(*
SPDX-FileCopyrightText: © 2026 Oleksandr Tiutyk <trofimich@gmail.com>
SPDX-License-Identifier: MIT
License: https://opensource.org/license/mit
*)

(*!
<summary>
Beckhoff EL1004: 4-channel digital input terminal (24 V DC, 3 ms filter).
</summary>
<description>
Process image mapping structure for the EL1004 EtherCAT terminal with 4 discrete 24 V DC inputs.
When used for I/O, link located fields or their containing buffers to the matching selected PDOs.
The record is not a packed wire buffer; compiler padding is not part of the device specification.
Unlinked/default values do not prove valid I/O. The caller evaluates bus/channel validity before use.
Use one owner task per instance and externally synchronize other access; multi-field snapshots are not atomic.
Copies store data without creating hardware links. Keep borrowed field references valid while consumers are bound.
This passive record performs no validation, synchronization, configuration or protocol advancement.
</description>
*)
TYPE EL1004 :
STRUCT
	Ch1 AT %I* : BOOL;
	Ch2 AT %I* : BOOL;
	Ch3 AT %I* : BOOL;
	Ch4 AT %I* : BOOL;
END_STRUCT
END_TYPE

(* stored: Version 1.1.0.1, ProductVersion 3.1.4026.20
   DUT EL1004: Id {0d568fa3-9585-4d01-884b-fcda27f7783b} *)
